// Core §3.15 — networked smart device: session + mandatory link supervision.
INTERFACE I_DeviceConnector EXTENDS I_Module

METHOD Connect : BOOL
END_METHOD

METHOD Disconnect : BOOL
END_METHOD

// timestamp of last healthy heartbeat (Core §2.7)
PROPERTY LastSeen : DT
GET
END_GET
END_PROPERTY

// session up AND heartbeat healthy (Core §3.15.2)
PROPERTY Linked : BOOL
GET
END_GET
END_PROPERTY

// first-out link/protocol reason when not Linked
PROPERTY LinkReason : ST_Diagnostic
GET
END_GET
END_PROPERTY

END_INTERFACE

(* stored: Version 1.1.0.1, ProductVersion 3.1.4024.12
   Itf I_DeviceConnector: Id {6fceefb2-967c-4678-aea0-3e92b415e1dc}
   Method Connect: Id {45bbd8bb-8dd5-4e83-ae93-5bf4e5a0c7db}
   Method Disconnect: Id {8dedb901-a8a0-42b5-81bb-e23b761e875a}
   Property LastSeen: Id {8e41e9fe-9bf7-492a-af08-cc128968f6ff}
   Get Get: Id {98665b6a-981c-4f36-9fa3-effae047b0f2}
   Property Linked: Id {620ccd86-b30b-4c4f-b5c1-8cf449315c82}
   Get Get: Id {84ba559a-e85d-4179-9085-289dfde2cab3}
   Property LinkReason: Id {7aed6a54-47ac-479a-b4ff-631e3098864a}
   Get Get: Id {13cb7ebe-df78-49a9-9c97-4d712c4cd5a1} *)
